      ;FOLD t9 ( EIN ) = STOP ;%{SE}%MKUKATPVW %CVW_SPS %VTSTOP %P 2:t9 ( EIN ) = STOP, 3: TSTOP
         VW(#SET_TIME,TRUE,9,1,0)
      ;ENDFOLD
      ;FOLD -- RSK Fehlerausgabe Kraftaufbau -- ;%{SE}%MKUKATPVW %CVW_COM %VCOMMENT %P 2:-- RSK Fehlerausgabe Kraftaufbau --, 3: VW_COMMENT
      ;ENDFOLD
      ;FOLD F325 = T9 ;%{SE}%MKUKATPVW %CVW_SPS %VBOASG %P 2:F325 = T9, 3: BOASG
         $FLAG[325] = $TIMER_FLAG[9]
      ;ENDFOLD
      ;FOLD -- KF1 abschalten bei Fehler -- ;%{SE}%MKUKATPVW %CVW_COM %VCOMMENT %P 2:-- KF1 abschalten bei Fehler --, 3: VW_COMMENT
      ;ENDFOLD
      ;FOLD A834 = !T7 & !T9 ;%{SE}%MKUKATPVW %CVW_SPS %VBOASG %P 2:A834 = !T7 & !T9, 3: BOASG
         $OUT[834] = NOT $TIMER_FLAG[7] AND NOT $TIMER_FLAG[9]
      ;ENDFOLD
      ;FOLD A858 = !T7 & !T9 ;%{SE}%MKUKATPVW %CVW_SPS %VBOASG %P 2:A858 = !T7 & !T9, 3: BOASG
         $OUT[858] = NOT $TIMER_FLAG[7] AND NOT $TIMER_FLAG[9]
      ;ENDFOLD
      ;FOLD A859 = !T7 & !T9 ;%{SE}%MKUKATPVW %CVW_SPS %VBOASG %P 2:A859 = !T7 & !T9, 3: BOASG
         $OUT[859] = NOT $TIMER_FLAG[7] AND NOT $TIMER_FLAG[9]
      ;ENDFOLD
      ;FOLD -- Warte Fraesen fertig oder Timeout -- ;%{SE}%MKUKATPVW %CVW_COM %VCOMMENT %P 2:-- Warte Fraesen fertig oder Timeout --, 3: VW_COMMENT
      ;ENDFOLD
      ;FOLD Schritt 281 = (F79 & F98 + F78 & F94 & !F287 + F78 & F96 & F287 + T7 + T9) & A4039  ;%{SE}%MKUKATPVW %CVW_SPS %VST_CON %P 2:Schritt 281 = (F79 & F98 + F78 & F94 & !F287 + F78 & F96 & F287 + T7 + T9) & A4039 , 3: ST_CON
         IF ($FLAG[79] AND $FLAG[98] OR $FLAG[78] AND $FLAG[94] AND NOT $FLAG[287] OR $FLAG[78] AND $FLAG[96] AND $FLAG[287] OR $TIMER_FLAG[7] OR $TIMER_FLAG[9]) AND $OUT[4039] THEN
            PREVSTEP = $APP_INT[5]
            $APP_INT[5] = 281
         ENDIF
      ;ENDFOLD
   ;ENDFOLD
   ;FOLD SCHRITT 281 -- ROB STP1 SZ1 # Ende -- ;%{P}%MKUKATPVW,%CSTEP,%VST_NR,%P 1:SCHRITT, 2:281, 3: ROB STP1 SZ1 # Ende
      ;FOLD ;%{H}
         Case 281
      ;ENDFOLD
      ;FOLD t7 ( EIN ) = STOP ;%{SE}%MKUKATPVW %CVW_SPS %VTSTOP %P 2:t7 ( EIN ) = STOP, 3: TSTOP
         VW(#SET_TIME,TRUE,7,1,0)
      ;ENDFOLD
      ;FOLD -- Wartezeit Programmwechsel SK -- ;%{SE}%MKUKATPVW %CVW_COM %VCOMMENT %P 2:-- Wartezeit Programmwechsel SK --, 3: VW_COMMENT
      ;ENDFOLD
      ;FOLD t8 ( EIN ) = -1[1/10Sek] ;%{SE}%MKUKATPVW %CVW_SPS %VTASG %P 2:t8 ( EIN ) = -1[1/10Sek], 3: TASG
         VW(#SET_TIME,TRUE,8,0,-1)
      ;ENDFOLD
      ;FOLD -- EZ1/SP1 SZ1 oeffnen -- ;%{SE}%MKUKATPVW %CVW_COM %VCOMMENT %P 2:-- EZ1/SP1 SZ1 oeffnen --, 3: VW_COMMENT
      ;ENDFOLD
      ;FOLD A718 = AUS ;%{SE}%MKUKATPVW %CVW_SPS %VBOASG %P 2:A718 = AUS, 3: BOASG
         $OUT[718] = FALSE
      ;ENDFOLD
      ;FOLD A717 = EIN ;%{SE}%MKUKATPVW %CVW_SPS %VBOASG %P 2:A717 = EIN, 3: BOASG
         $OUT[717] = TRUE
      ;ENDFOLD
      ;FOLD -- KF1 Ausblasen -- ;%{SE}%MKUKATPVW %CVW_COM %VCOMMENT %P 2:-- KF1 Ausblasen --, 3: VW_COMMENT
      ;ENDFOLD
      ;FOLD A835 = !F289 ;%{SE}%MKUKATPVW %CVW_SPS %VBOASG %P 2:A835 = !F289, 3: BOASG
         $OUT[835] = NOT $FLAG[289]
      ;ENDFOLD
      ;FOLD A859 = A835 & F289 ;%{SE}%MKUKATPVW %CVW_SPS %VBOASG %P 2:A859 = A835 & F289, 3: BOASG
         $OUT[859] = $OUT[835] AND $FLAG[289]
      ;ENDFOLD
      ;FOLD -- RSK Sammelstoerung -- ;%{SE}%MKUKATPVW %CVW_COM %VCOMMENT %P 2:-- RSK Sammelstoerung --, 3: VW_COMMENT
      ;ENDFOLD
      ;FOLD F329 = T7 + T9 ;%{SE}%MKUKATPVW %CVW_SPS %VBOASG %P 2:F329 = T7 + T9, 3: BOASG
         $FLAG[329] = $TIMER_FLAG[7] OR $TIMER_FLAG[9]
      ;ENDFOLD
      ;FOLD -- Hilfsflag Startfraesen -- ;%{SE}%MKUKATPVW %CVW_COM %VCOMMENT %P 2:-- Hilfsflag Startfraesen --, 3: VW_COMMENT
      ;ENDFOLD
      ;FOLD F96 = (F96 & F78 + F98 & F79) & F287 ;%{SE}%MKUKATPVW %CVW_SPS %VBOASG %P 2:F96 = (F96 & F78 + F98 & F79) & F287, 3: BOASG
         $FLAG[96] = ($FLAG[96] AND $FLAG[78] OR $FLAG[98] AND $FLAG[79]) AND $FLAG[287]
      ;ENDFOLD
      ;FOLD F98 = !F130 & F98 + F130 & F287 & F98 ;%{SE}%MKUKATPVW %CVW_SPS %VBOASG %P 2:F98 = !F130 & F98 + F130 & F287 & F98, 3: BOASG
         $FLAG[98] = NOT $FLAG[130] AND $FLAG[98] OR $FLAG[130] AND $FLAG[287] AND $FLAG[98]
      ;ENDFOLD
      ;FOLD F287 = F78 + F79 & F130 ;%{SE}%MKUKATPVW %CVW_SPS %VBOASG %P 2:F287 = F78 + F79 & F130, 3: BOASG
         $FLAG[287] = $FLAG[78] OR $FLAG[79] AND $FLAG[130]
      ;ENDFOLD
      ;FOLD -- Neues Fraesprogramm und Zaehler ruecksetzen -- ;%{SE}%MKUKATPVW %CVW_COM %VCOMMENT %P 2:-- Neues Fraesprogramm und Zaehler ruecksetzen --, 3: VW_COMMENT
      ;ENDFOLD
      ;FOLD F270 = F96 & F732 ;%{SE}%MKUKATPVW %CVW_SPS %VBOASG %P 2:F270 = F96 & F732, 3: BOASG
         $FLAG[270] = $FLAG[96] AND $FLAG[732]
      ;ENDFOLD
      ;FOLD bin3 ( F732 ) = 36 ;%{SE}%MKUKATPVW %CVW_SPS %VARIASG %P 2:bin3 ( F732 ) = 36, 3: ARIASG
         VW(#BINOUT,$FLAG[732],3,36)
      ;ENDFOLD
      ;FOLD i4 ( F270 ) = i45 ;%{SE}%MKUKATPVW %CVW_SPS %VARIASG %P 2:i4 ( F270 ) = i45, 3: ARIASG
         VW(#COUNTER,$FLAG[270],4,$COUNT_I[45])
      ;ENDFOLD
      ;FOLD -- Wiederholung beim Startfraesen -- ;%{SE}%MKUKATPVW %CVW_COM %VCOMMENT %P 2:-- Wiederholung beim Startfraesen --, 3: VW_COMMENT
      ;ENDFOLD
      ;FOLD Schritt 276 = E717 & !E718 & (F78 & !F96 + F79 & F130 & !F96) & !F329 & A4039  ;%{SE}%MKUKATPVW %CVW_SPS %VST_CON %P 2:Schritt 276 = E717 & !E718 & (F78 & !F96 + F79 & F130 & !F96) & !F329 & A4039 , 3: ST_CON
         IF $IN[717] AND NOT $IN[718] AND ($FLAG[78] AND NOT $FLAG[96] OR $FLAG[79] AND $FLAG[130] AND NOT $FLAG[96]) AND NOT $FLAG[329] AND $OUT[4039] THEN
            PREVSTEP = $APP_INT[5]
            $APP_INT[5] = 276
         ENDIF
      ;ENDFOLD
      ;FOLD -- Weiter wenn Fraesen fertig -- ;%{SE}%MKUKATPVW %CVW_COM %VCOMMENT %P 2:-- Weiter wenn Fraesen fertig --, 3: VW_COMMENT
      ;ENDFOLD
      ;FOLD Schritt 282 = E717 & !E718 & (F79 & F98 & (!F130 + F96) + F78 & F96 + F329) & A4039  ;%{SE}%MKUKATPVW %CVW_SPS %VST_CON %P 2:Schritt 282 = E717 & !E718 & (F79 & F98 & (!F130 + F96) + F78 & F96 + F329) & A4039 , 3: ST_CON
         IF $IN[717] AND NOT $IN[718] AND ($FLAG[79] AND $FLAG[98] AND (NOT $FLAG[130] OR $FLAG[96]) OR $FLAG[78] AND $FLAG[96] OR $FLAG[329]) AND $OUT[4039] THEN
            PREVSTEP = $APP_INT[5]
            $APP_INT[5] = 282
         ENDIF
      ;ENDFOLD
      ;FOLD -- Weiter bei Fehler -- ;%{SE}%MKUKATPVW %CVW_COM %VCOMMENT %P 2:-- Weiter bei Fehler --, 3: VW_COMMENT
      ;ENDFOLD
      ;FOLD Schritt 284 = F325 & (E26 + E27) & A4039  ;%{SE}%MKUKATPVW %CVW_SPS %VST_CON %P 2:Schritt 284 = F325 & (E26 + E27) & A4039 , 3: ST_CON
         IF $FLAG[325] AND ($IN[26] OR $IN[27]) AND $OUT[4039] THEN
            PREVSTEP = $APP_INT[5]
            $APP_INT[5] = 284
         ENDIF
      ;ENDFOLD
   ;ENDFOLD
   ;FOLD SCHRITT 282 -- ROB EZ1/SP1 SZ1 -- ;%{P}%MKUKATPVW,%CSTEP,%VST_NR,%P 1:SCHRITT, 2:282, 3: ROB EZ1/SP1 SZ1
      ;FOLD ;%{H}
         Case 282
      ;ENDFOLD
      ;FOLD F270 = AUS ;%{SE}%MKUKATPVW %CVW_SPS %VBOASG %P 2:F270 = AUS, 3: BOASG
         $FLAG[270] = FALSE
      ;ENDFOLD
      ;FOLD A717 = AUS ;%{SE}%MKUKATPVW %CVW_SPS %VBOASG %P 2:A717 = AUS, 3: BOASG
         $OUT[717] = FALSE
      ;ENDFOLD
      ;FOLD -- KF1 abschalten -- ;%{SE}%MKUKATPVW %CVW_COM %VCOMMENT %P 2:-- KF1 abschalten --, 3: VW_COMMENT
      ;ENDFOLD
      ;FOLD A834 = AUS ;%{SE}%MKUKATPVW %CVW_SPS %VBOASG %P 2:A834 = AUS, 3: BOASG
         $OUT[834] = FALSE
      ;ENDFOLD
      ;FOLD A858 = AUS ;%{SE}%MKUKATPVW %CVW_SPS %VBOASG %P 2:A858 = AUS, 3: BOASG
         $OUT[858] = FALSE
      ;ENDFOLD
      ;FOLD A859 = AUS ;%{SE}%MKUKATPVW %CVW_SPS %VBOASG %P 2:A859 = AUS, 3: BOASG
         $OUT[859] = FALSE
      ;ENDFOLD
      ;FOLD bin3 ( !F329 ) = 1 ;%{SE}%MKUKATPVW %CVW_SPS %VARIASG %P 2:bin3 ( !F329 ) = 1, 3: ARIASG
         VW(#BINOUT,NOT $FLAG[329],3,1)
      ;ENDFOLD
      ;FOLD Schritt 283 = T8 & A4039  ;%{SE}%MKUKATPVW %CVW_SPS %VST_CON %P 2:Schritt 283 = T8 & A4039 , 3: ST_CON
         IF $TIMER_FLAG[8] AND $OUT[4039] THEN
            PREVSTEP = $APP_INT[5]
            $APP_INT[5] = 283
         ENDIF
      ;ENDFOLD
   ;ENDFOLD
   ;FOLD SCHRITT 283 -- ROB EZ1/SP1 SZ1 -- ;%{P}%MKUKATPVW,%CSTEP,%VST_NR,%P 1:SCHRITT, 2:283, 3: ROB EZ1/SP1 SZ1
      ;FOLD ;%{H}
         Case 283
      ;ENDFOLD
      ;FOLD -- Quitt. Fraesen SK1 -- ;%{SE}%MKUKATPVW %CVW_COM %VCOMMENT %P 2:-- Quitt. Fraesen SK1 --, 3: VW_COMMENT
      ;ENDFOLD
      ;FOLD A786 = !F329 & !F322 ;%{SE}%MKUKATPVW %CVW_SPS %VBOASG %P 2:A786 = !F329 & !F322, 3: BOASG
         $OUT[786] = NOT $FLAG[329] AND NOT $FLAG[322]
      ;ENDFOLD
      ;FOLD Schritt 284 = (!E786 & E787 & !E788 + F329) & A4039  ;%{SE}%MKUKATPVW %CVW_SPS %VST_CON %P 2:Schritt 284 = (!E786 & E787 & !E788 + F329) & A4039 , 3: ST_CON
         IF (NOT $IN[786] AND $IN[787] AND NOT $IN[788] OR $FLAG[329]) AND $OUT[4039] THEN
            PREVSTEP = $APP_INT[5]
            $APP_INT[5] = 284
         ENDIF
      ;ENDFOLD
   ;ENDFOLD
   ;FOLD SCHRITT 284 -- ROB EZ1/SP1 SZ1 # Ende -- ;%{P}%MKUKATPVW,%CSTEP,%VST_NR,%P 1:SCHRITT, 2:284, 3: ROB EZ1/SP1 SZ1 # Ende
      ;FOLD ;%{H}
         Case 284
      ;ENDFOLD
      ;FOLD -- KF1 Ausblasen -- ;%{SE}%MKUKATPVW %CVW_COM %VCOMMENT %P 2:-- KF1 Ausblasen --, 3: VW_COMMENT
      ;ENDFOLD
      ;FOLD A835 = AUS ;%{SE}%MKUKATPVW %CVW_SPS %VBOASG %P 2:A835 = AUS, 3: BOASG
         $OUT[835] = FALSE
      ;ENDFOLD
      ;FOLD A859 = A835 ;%{SE}%MKUKATPVW %CVW_SPS %VBOASG %P 2:A859 = A835, 3: BOASG
         $OUT[859] = $OUT[835]
      ;ENDFOLD
      ;FOLD F91 = !E786 & E787 & !E788 & !F322 & !F325 & !F329 ;%{SE}%MKUKATPVW %CVW_SPS %VBOASG %P 2:F91 = !E786 & E787 & !E788 & !F322 & !F325 & !F329, 3: BOASG
         $FLAG[91] = NOT $IN[786] AND $IN[787] AND NOT $IN[788] AND NOT $FLAG[322] AND NOT $FLAG[325] AND NOT $FLAG[329]
      ;ENDFOLD
      ;FOLD Schritt 272 = (F322 + F325 + F329) & (E26 + E27) & A4039  ;%{SE}%MKUKATPVW %CVW_SPS %VST_CON %P 2:Schritt 272 = (F322 + F325 + F329) & (E26 + E27) & A4039 , 3: ST_CON
         IF ($FLAG[322] OR $FLAG[325] OR $FLAG[329]) AND ($IN[26] OR $IN[27]) AND $OUT[4039] THEN
            PREVSTEP = $APP_INT[5]
            $APP_INT[5] = 272
         ENDIF
      ;ENDFOLD
      ;FOLD Schritt 1 = F91 & !F322 & !F325 & !F329 & A4039  ;%{SE}%MKUKATPVW %CVW_SPS %VST_CON %P 2:Schritt 1 = F91 & !F322 & !F325 & !F329 & A4039 , 3: ST_CON
         IF $FLAG[91] AND NOT $FLAG[322] AND NOT $FLAG[325] AND NOT $FLAG[329] AND $OUT[4039] THEN
            PREVSTEP = $APP_INT[5]
            $APP_INT[5] = 1
         ENDIF
      ;ENDFOLD
   ;ENDFOLD
   ; FOLD ;%{H}
   DEFAULT
   HMeldung ("StepNotAvailable")
   $APP_INT[5]=1
   ENDSWITCH
   END
   DEF HMeldung (Meld[]:IN)
     CHAR Meld[]
     DECL KrlMsg_T Msg
     DECL KrlMsgPar_T Par[3]
     DECL KrlMsgOpt_T Opt
     INT nHandle
     BOOL dummy
     dummy=STRCOPY(Msg.Msg_txt[],Meld[])
     Msg.Modul[]="MAKROSTEP"
     Msg.Nr=110
     Par[1].Par_type=#Value
     Par[1].Par_Int = PREVSTEP
     Opt = {VL_Stop TRUE, Clear_P_Reset TRUE, Log_To_DB FALSE}
     nHandle = Set_KrlMsg (#Notify, Msg, Par[], Opt)
     WAIT SEC 0.2
END
; ENDFOLD
